FUNCTION_BLOCK FB_ControlSignal
VAR_INPUT
	fUFF : LREAL;
	fPID : LREAL;
	bEnableU : BOOL;
	fQMaxUp 	: LREAL; // Needs to be positive (22)
	fQMaxDown 	: LREAL; // Needs to be positive (15)
	fDeadUp		: LREAL; // Needs to be positive (0.155)
	fDeadDown 	: LREAL; // Needs to be positive (0.18)
	
	fXDotRef	: LREAL;
	fError		: LREAL;
END_VAR
VAR_OUTPUT
	fU : LREAL;
END_VAR
VAR

	fUTemp : LREAL;
	fUTemp2 : LREAL;
	fUMax : LREAL := 0.9;
END_VAR

IF bEnableU THEN
	fUTemp := fUFF  - fPID;
	
	// Deadband compensation
	IF (fXDotRef > 0 OR fXDotRef < 0) OR fError > 0.002 THEN
		IF fUTemp <= 0.0 THEN	// Upwards
			fUTemp2 := fUTemp - fDeadUp;
		ELSIF fUTemp > 0.0 THEN // Downwards
			fUTemp2 := fUTemp + fDeadDown;
		END_IF
		
		IF fUTemp2 >= fUMax THEN
			fU := fUMax;
		ELSIF fUTemp2 <= -fUMax THEN
			fU := -fUMax;
		ELSE
			fU := fUTemp2;
		END_IF
	ELSE
		fU := 0.0;
	END_IF
END_IF

END_FUNCTION_BLOCK

(* stored: Version 1.1.0.1, ProductVersion 3.1.4024.12
   POU FB_ControlSignal: Id {5ec98e7b-f91c-4803-9df2-1eb6eb99ed16}, SpecialFunc None *)
